(* CODESYS project refactoreddoworking.project
   CompiledLibraryCompatibilityVersion: LeadSysStudio V3.5 SP15 Patch 4
   Title: MC500_EtherCAT_axis_motion

Project tree, tasks and I/O mapping:
  Device : MC508, Leadshine Technology Co., Ltd., order no. 508101, version 3.5.15.40
      settings: RetainMode = 0; RetainStartAddr = 20480; RetainEndAddr = 524288; RetainSize = 524288
    application Application
      libraries: Standard, * (System); LS_ModbusMasterlib, 0.0.0.2 (Leadshine Technology Co.Ltd)
      task MainTask (cyclic, interval 4000 µs, priority 1) calls EtherCAT_Master_Leadshine_A.EtherCAT_Task, PLC_PRG
      global variables GVL_Shared
      program MainSeq [SFC]: A_Idle, A_HomeXY, A_GridCalc, A_GriddleDwell, A_MoveToPick, A_Grip, A_MoveToPlace, A_Release, A_NextOrDone, A_Park, A_Wait, A_Settle, A_Error, A_Hold, A_ZDownPick, A_ZUp, A_ZDownPlace, A_ZUpAfter, A_ZWait
      program PLC_PRG [CFC]
      program Inputs [LD]
      program Motion [CFC]
      function block GridCalc [ST]
    Resource Usage
    Network Configuration
      LocalBus Config
    Device Diagnose
    LocalBus_Master_Module : LocalBus Master, Leadshine Technology Co., Ltd., version 3.5.15.40
    High_Speed_IO_Module : High Speed IO, Leadshine Technology Co., Ltd., version 3.5.15.40
        unmapped channels: Genral_IO_IN, Genral_IO_Out
    SoftMotion General Axis Pool
    EtherCAT_Master_Leadshine_A : EtherCAT Master SoftMotion, 3S - Smart Software Solutions GmbH, version 3.5.15.30
        settings: NetworkName = 'ecat'; SelectNetworkByName = TRUE
      CS3E_D1008 : CS3E-D1008(COE), Leadshine Technology Co.,Ltd., order no. CS3E-D1008, version Revision=16#00000001
          settings: DC sync0 cycletime = 4000; DC sync1 cycletime = 4000; Number of SDO = 6; Homing method.Index = 16#6098; Homing method.Subindex = 16#00; Homing method.Value = 17; Homing method.Size = 8; Homing method.AbortIfError = FALSE; Homing method.JumpToLine = FALSE; Homing method.Line = 0; Homing method.CompleteAccess = FALSE; Homing velocity (fast).Index = 16#6099; Homing velocity (fast).Subindex = 16#01; Homing velocity (fast).Value = 2000; Homing velocity (fast).Size = 32; Homing velocity (fast).AbortIfError = FALSE; Homing velocity (fast).JumpToLine = FALSE; Homing velocity (fast).Line = 0; Homing velocity (fast).CompleteAccess = FALSE; Homing velocity (slow).Index = 16#6099; Homing velocity (slow).Subindex = 16#02; Homing velocity (slow).Value = 300; Homing velocity (slow).Size = 32; Homing velocity (slow).AbortIfError = FALSE; Homing velocity (slow).JumpToLine = FALSE; Homing velocity (slow).Line = 0; Homing velocity (slow).CompleteAccess = FALSE; Homing acceleration.Index = 16#609A; Homing acceleration.Subindex = 16#00; Homing acceleration.Value = 5000; Homing acceleration.Size = 32; Homing acceleration.AbortIfError = FALSE; Homing acceleration.JumpToLine = FALSE; Homing acceleration.Line = 0; Homing acceleration.CompleteAccess = FALSE; Homing offset.Index = 16#607C; Homing offset.Subindex = 16#00; Homing offset.Value = 0; Homing offset.Size = 32; Homing offset.AbortIfError = FALSE;
            Homing offset.JumpToLine = FALSE; Homing offset.Line = 0; Homing offset.CompleteAccess = FALSE
          input  yAxis_LastError : UINT  // Last Error Code
          unmapped channels: Control Word, Profile Target Position, Touch Probe Function, Status Word, Modes of Operation display, Position Actual Value, Touch Probe Status, Touch Probe 1 Positive Value, Digital Inputs
        yAxis : Axis, 3S - Smart Software Solutions GmbH, order no. 0, version 4.6.1.0
            settings: wDriveID = 0; dwRatioTechUnitsDenom = 20; eRampType = 3; Number of pulses for one revolution = 4000; The displacement for one revolution of the workbench = 100; Gear ratio molecule = 10; Gear ratio denominator = 10; Home velocity = 100; Home Creep speed = 15.000; Home acceleration = 250; Home position offset = 0; Home velocitySDO = 2000; Home Creep speedSDO = 300; Home position offsetSDO = 0; ScalingIncs = 4000; AdrOffset_8010 = 16; BitOffset_8010 = 0; BitLength_8010 = 16; Address_8010 = '%QW8'; Type_8010 = 'UINT'; AddressPointer_8010 = ADR(%QW8); AdrOffset_8020 = 20; BitOffset_8020 = 0; BitLength_8020 = 32; Address_8020 = '%QD5'; Type_8020 = 'DINT'; AddressPointer_8020 = ADR(%QD5); AdrOffset_8030 = 4294967295; BitOffset_8030 = 0; BitLength_8030 = 0; Address_8030 = ''; Type_8030 = ''; AddressPointer_8030 = 0; AdrOffset_8040 = 4294967295; BitOffset_8040 = 0; BitLength_8040 = 0; Address_8040 = ''; Type_8040 = ''; AddressPointer_8040 = 0; AdrOffset_8050 = 4294967295;
              BitOffset_8050 = 0; BitLength_8050 = 0; Address_8050 = ''; Type_8050 = ''; AddressPointer_8050 = 0; AdrOffset_8060 = 24; BitOffset_8060 = 0; BitLength_8060 = 16; Address_8060 = '%QW12'; Type_8060 = 'UINT'; AddressPointer_8060 = ADR(%QW12); AdrOffset_8070 = 4294967295; BitOffset_8070 = 0; BitLength_8070 = 0; Address_8070 = ''; Type_8070 = ''; AddressPointer_8070 = 0; AdrOffset_8080 = 4294967295; BitOffset_8080 = 0; BitLength_8080 = 0; Address_8080 = ''; Type_8080 = ''; AddressPointer_8080 = 0; AdrOffset_8090 = 4294967295; BitOffset_8090 = 0; BitLength_8090 = 0; Address_8090 = ''; Type_8090 = ''; AddressPointer_8090 = 0; AdrOffset_8510 = 30; BitOffset_8510 = 0; BitLength_8510 = 16; Address_8510 = '%IW15'; Type_8510 = 'UINT'; AddressPointer_8510 = ADR(%IW15); AdrOffset_8520 = 36; BitOffset_8520 = 0; BitLength_8520 = 32; Address_8520 = '%ID9'; Type_8520 = 'DINT';
              AddressPointer_8520 = ADR(%ID9); AdrOffset_8530 = 4294967295; BitOffset_8530 = 0; BitLength_8530 = 0; Address_8530 = ''; Type_8530 = ''; AddressPointer_8530 = 0; AdrOffset_8540 = 4294967295; BitOffset_8540 = 0; BitLength_8540 = 0; Address_8540 = ''; Type_8540 = ''; AddressPointer_8540 = 0; AdrOffset_8550 = 32; BitOffset_8550 = 0; BitLength_8550 = 8; Address_8550 = '%IB32'; Type_8550 = 'SINT'; AddressPointer_8550 = ADR(%IB32); AdrOffset_8560 = 48; BitOffset_8560 = 0; BitLength_8560 = 32; Address_8560 = '%ID12'; Type_8560 = 'UDINT'; AddressPointer_8560 = ADR(%ID12); AdrOffset_8570 = 40; BitOffset_8570 = 0; BitLength_8570 = 16; Address_8570 = '%IW20'; Type_8570 = 'UINT'; AddressPointer_8570 = ADR(%IW20); AdrOffset_8580 = 44; BitOffset_8580 = 0; BitLength_8580 = 32; Address_8580 = '%ID11'; Type_8580 = 'DINT'; AddressPointer_8580 = ADR(%ID11); AdrOffset_8590 = 4294967295; BitOffset_8590 = 0; BitLength_8590 = 0;
              Address_8590 = ''; Type_8590 = ''; AddressPointer_8590 = 0; AdrOffset_8600 = 4294967295; BitOffset_8600 = 0; BitLength_8600 = 0; Address_8600 = ''; Type_8600 = ''; AddressPointer_8600 = 0; AdrOffset_8600 = 4294967295; BitOffset_8600 = 0; BitLength_8600 = 0; Address_8610 = ''; Type_8610 = ''; AddressPointer_8610 = 0; AdrOffset_8620 = 4294967295; BitOffset_8620 = 0; BitLength_8620 = 0; Address_8620 = ''; Type_8620 = ''; AddressPointer_8620 = 0; Home accelerationSDO = 5000
      CS3E_D1008_1 : CS3E-D1008(COE), Leadshine Technology Co.,Ltd., order no. CS3E-D1008, version Revision=16#00000001
          settings: DC sync0 cycletime = 4000; DC sync1 cycletime = 4000; Number of SDO = 6; Homing method.Index = 16#6098; Homing method.Subindex = 16#00; Homing method.Value = 17; Homing method.Size = 8; Homing method.AbortIfError = FALSE; Homing method.JumpToLine = FALSE; Homing method.Line = 0; Homing method.CompleteAccess = False; Homing velocity (fast).Index = 16#6099; Homing velocity (fast).Subindex = 16#01; Homing velocity (fast).Value = 2000; Homing velocity (fast).Size = 32; Homing velocity (fast).AbortIfError = FALSE; Homing velocity (fast).JumpToLine = FALSE; Homing velocity (fast).Line = 0; Homing velocity (fast).CompleteAccess = False; Homing velocity (slow).Index = 16#6099; Homing velocity (slow).Subindex = 16#02; Homing velocity (slow).Value = 300; Homing velocity (slow).Size = 32; Homing velocity (slow).AbortIfError = FALSE; Homing velocity (slow).JumpToLine = FALSE; Homing velocity (slow).Line = 0; Homing velocity (slow).CompleteAccess = False; Homing acceleration.Index = 16#609A; Homing acceleration.Subindex = 16#00; Homing acceleration.Value = 5000; Homing acceleration.Size = 32; Homing acceleration.AbortIfError = FALSE; Homing acceleration.JumpToLine = FALSE; Homing acceleration.Line = 0; Homing acceleration.CompleteAccess = False; Homing offset.Index = 16#607C; Homing offset.Subindex = 16#00; Homing offset.Value = 0; Homing offset.Size = 32; Homing offset.AbortIfError = FALSE;
            Homing offset.JumpToLine = FALSE; Homing offset.Line = 0; Homing offset.CompleteAccess = False
          input  XAXIS_LastError : UINT  // Last Error Code
          unmapped channels: Control Word, Profile Target Position, Touch Probe Function, Status Word, Modes of Operation display, Position Actual Value, Touch Probe Status, Touch Probe 1 Positive Value, Digital Inputs
        XAXIS : Axis, 3S - Smart Software Solutions GmbH, order no. 0, version 4.6.1.0
            settings: dwRatioTechUnitsDenom = 20; Commisioning.smci.Distance = 110; Commisioning.smci.Velocity = 100; Gear ratio molecule = 500; Gear ratio denominator = 500; Home velocity = 100; Home Creep speed = 15; Home acceleration = 250; Home position offset = 0; Home velocitySDO = 2000; Home Creep speedSDO = 300; Home position offsetSDO = 0; ScalingIncs = 4000; InvertDirection = False; AdrOffset_8010 = 4; BitOffset_8010 = 0; BitLength_8010 = 16; Address_8010 = '%QW2'; Type_8010 = 'UINT'; AddressPointer_8010 = ADR(%QW2); AdrOffset_8020 = 8; BitOffset_8020 = 0; BitLength_8020 = 32; Address_8020 = '%QD2'; Type_8020 = 'DINT'; AddressPointer_8020 = ADR(%QD2); AdrOffset_8030 = 4294967295; BitOffset_8030 = 0; BitLength_8030 = 0; Address_8030 = ''; Type_8030 = ''; AddressPointer_8030 = 0; AdrOffset_8040 = 4294967295; BitOffset_8040 = 0; BitLength_8040 = 0; Address_8040 = ''; Type_8040 = ''; AddressPointer_8040 = 0; AdrOffset_8050 = 4294967295; BitOffset_8050 = 0;
              BitLength_8050 = 0; Address_8050 = ''; Type_8050 = ''; AddressPointer_8050 = 0; AdrOffset_8060 = 12; BitOffset_8060 = 0; BitLength_8060 = 16; Address_8060 = '%QW6'; Type_8060 = 'UINT'; AddressPointer_8060 = ADR(%QW6); AdrOffset_8070 = 4294967295; BitOffset_8070 = 0; BitLength_8070 = 0; Address_8070 = ''; Type_8070 = ''; AddressPointer_8070 = 0; AdrOffset_8080 = 4294967295; BitOffset_8080 = 0; BitLength_8080 = 0; Address_8080 = ''; Type_8080 = ''; AddressPointer_8080 = 0; AdrOffset_8090 = 4294967295; BitOffset_8090 = 0; BitLength_8090 = 0; Address_8090 = ''; Type_8090 = ''; AddressPointer_8090 = 0; AdrOffset_8510 = 6; BitOffset_8510 = 0; BitLength_8510 = 16; Address_8510 = '%IW3'; Type_8510 = 'UINT'; AddressPointer_8510 = ADR(%IW3); AdrOffset_8520 = 12; BitOffset_8520 = 0; BitLength_8520 = 32; Address_8520 = '%ID3'; Type_8520 = 'DINT'; AddressPointer_8520 = ADR(%ID3);
              AdrOffset_8530 = 4294967295; BitOffset_8530 = 0; BitLength_8530 = 0; Address_8530 = ''; Type_8530 = ''; AddressPointer_8530 = 0; AdrOffset_8540 = 4294967295; BitOffset_8540 = 0; BitLength_8540 = 0; Address_8540 = ''; Type_8540 = ''; AddressPointer_8540 = 0; AdrOffset_8550 = 8; BitOffset_8550 = 0; BitLength_8550 = 8; Address_8550 = '%IB8'; Type_8550 = 'SINT'; AddressPointer_8550 = ADR(%IB8); AdrOffset_8560 = 24; BitOffset_8560 = 0; BitLength_8560 = 32; Address_8560 = '%ID6'; Type_8560 = 'UDINT'; AddressPointer_8560 = ADR(%ID6); AdrOffset_8570 = 16; BitOffset_8570 = 0; BitLength_8570 = 16; Address_8570 = '%IW8'; Type_8570 = 'UINT'; AddressPointer_8570 = ADR(%IW8); AdrOffset_8580 = 20; BitOffset_8580 = 0; BitLength_8580 = 32; Address_8580 = '%ID5'; Type_8580 = 'DINT'; AddressPointer_8580 = ADR(%ID5); AdrOffset_8590 = 4294967295; BitOffset_8590 = 0; BitLength_8590 = 0; Address_8590 = '';
              Type_8590 = ''; AddressPointer_8590 = 0; AdrOffset_8600 = 4294967295; BitOffset_8600 = 0; BitLength_8600 = 0; Address_8600 = ''; Type_8600 = ''; AddressPointer_8600 = 0; AdrOffset_8600 = 4294967295; BitOffset_8600 = 0; BitLength_8600 = 0; Address_8610 = ''; Type_8610 = ''; AddressPointer_8610 = 0; AdrOffset_8620 = 4294967295; BitOffset_8620 = 0; BitLength_8620 = 0; Address_8620 = ''; Type_8620 = ''; AddressPointer_8620 = 0; Home accelerationSDO = 5000
    ModbusTCP_Slave_Device : Modbus TCP Slave, Leadshine Technology Co., Ltd., version 00.00.00.10
*)

// Device/Application/GVL_Shared
// =====================================================================
// GVL  "GVL_Shared"  — globals shared across the LD / CFC / SFC / ST POUs
// (Splitting one POU into four means the formerly-local VARs become globals
//  grouped by owner. Comment // [owner->reader] shows the data direction.)
// =====================================================================
VAR_GLOBAL
    // ---- AXIS REFERENCES (declared in your hardware config) ----
    // XAXIS, yAxis : AXIS_REF;   // already exist in the project

    // ============ COMMAND FLAGS : LD (Inputs) -> SFC ============
    pending_start   : BOOL := FALSE;
    
    pending_resume  : BOOL := FALSE;
   
    hmi_start       : BOOL := FALSE;   // HMI write
   
    sw_a            : BOOL := FALSE;    // HMI/soft button A
    sw_b            : BOOL := FALSE;    // HMI/soft button B

    // ============ MOTION REQUESTS : SFC -> CFC (Motion) =========
    gMoveExec    : BOOL := FALSE;          // drive LS_MoveXY.Exec
    gHomeExec    : BOOL := FALSE;          // drive MC_Home_1/2.Execute
    gStopExec    : BOOL := FALSE;          // drive MC_Stop_1/2.Execute
    TargetXY     : ARRAY[0..1] OF LREAL := [0.0, 0.0];
    drive_enable : BOOL := TRUE;           // MC_Power_*.Enable (set by Inputs/Pause)

    // ============ MOTION STATUS : CFC (Motion) -> SFC ===========
    gPowerOK   : BOOL := FALSE;            // MC_Power_1.Status AND MC_Power_2.Status
    gMoveDone  : BOOL := FALSE;            // LS_MoveXY.Done
    gMoveErr   : BOOL := FALSE;            // LS_MoveXY.Error 
    gMoveBusy  : BOOL := FALSE;            // LS_MoveXY.Busy
    gHomeDone  : BOOL := FALSE;            // MC_Home_1.Done AND MC_Home_2.Done
    gStopDone  : BOOL := FALSE;            // MC_Stop_1.Done AND MC_Stop_2.Done

    // ============ END EFFECTOR + STOP TUNING ====================
    end_effector AT %QX1.4 : BOOL := FALSE;   // LD coil
    QUICK_STOP_DECEL : LREAL := 3000.0;

    // ============ Z AXIS — MODBUS I/O (CS2RS-D1008) =============


    // ============ TRAY / GRID CONFIG (read by GridCalc) ========
    PICK_BASE_X    : LREAL := 145.0;
    PICK_BASE_Y    : LREAL := 45.0;
    PICK_SPACING_X : LREAL := 80.0;
    PICK_SPACING_Y : LREAL := 80.0;
    PLACE_BASE_X   : LREAL := 740.0;
    PLACE_BASE_Y   : LREAL := 116.0;
    PLACE_OFFSET_X : ARRAY[0..5] OF LREAL := [0.0, 70.0, -70.0, 70.0, -70.0, 0.0];
    PLACE_OFFSET_Y : ARRAY[0..5] OF LREAL := [0.0, 66.0, 66.0, 143.0, 143.0, 210.0];
    TRAY_COLS           : INT := 6;
    TRAY_ROWS           : INT := 4;
    TOTAL_PATTIES       : INT := 24;
    PATTIES_PER_GRIDDLE : INT := 6;
    GRIDDLE_COUNT       : INT := 4;

    // ============ GRID RESULTS (GridCalc -> SFC) ===============
    patty_index   : INT := 0;
    current_col   : INT := 0;
    current_row   : INT := 0;
    griddle_index : INT := 0;
    slot_index    : INT := 0;
    pick_x  : LREAL := 0.0;   pick_y  : LREAL := 0.0;
    place_x : LREAL := 0.0;   place_y : LREAL := 0.0;

    // ============ MODE / BOOKKEEPING ===========================
    TEST_LOOP_MODE : BOOL := TRUE;
    cycle_count    : UDINT := 0;
    cycle_complete : BOOL := FALSE;
    cycle_active   : BOOL := FALSE;
    paused         : BOOL := FALSE;
   
    
    

    // ============ TIMING CONSTANTS =============================

   
    XY_HOME_WAIT   : INT := 7500;
    xy_home_timer  : INT := 0;
	
	stop_request  : BOOL := FALSE;   // CYCLE-stop request (operator Stop button)
	holding       : BOOL := FALSE;   // TRUE while parked & held
	pending_reset : BOOL := FALSE;
	hmi_stop      : BOOL := FALSE;
	hmi_reset     : BOOL := FALSE;
	
	
	Z_DO_Down    AT %QX1.5 : BOOL := FALSE;   // pulse -> down path
	Z_InPos      AT %IX1.0 : BOOL;            // SO1 INP = positioning complete
	z_saw_moving : BOOL := FALSE;
	Z_Alarm AT %IX1.1 : BOOL;   // SO3 ALM (check polarity)
	z_wait_count   : INT  := 0;
    Z_MOVE_TIMEOUT : INT  := 2500;
	
	state : INT := 0;
	Z_Disable AT %QX1.3 : BOOL := FALSE;   // TRUE = disable Z drive; FALSE (default) = enabled
	Z_Trig AT %QX1.6 : BOOL := FALSE; 
	xy_moving : BOOL := FALSE;
	np_done : BOOL := FALSE;
END_VAR

// Device/Application/PLC_PRG
PROGRAM PLC_PRG
VAR
   
END_VAR

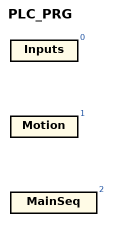
Inputs();
Motion();
MainSeq();

END_PROGRAM

// Device/Application/Inputs
PROGRAM Inputs
VAR
	btn_a AT %IX0.0 : BOOL;
    btn_b AT %IX0.1 : BOOL;
    rt_a : R_TRIG;
    rt_b : R_TRIG;
    edgeA : BOOL;                  
	edgeB : BOOL;
	btn_reset AT %IX0.2 : BOOL;   // physical Reset (wire later)
	rt_reset  : R_TRIG;
	edgeReset : BOOL;
END_VAR

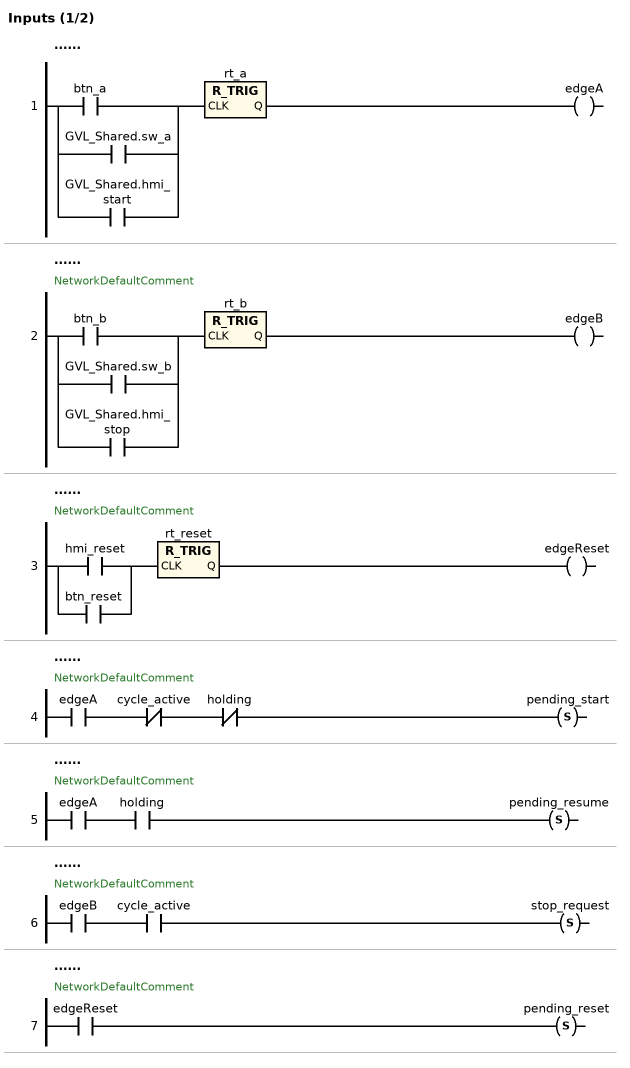
// NETWORK 1: ......
rt_a(CLK := btn_a OR GVL_Shared.sw_a OR GVL_Shared.hmi_start); // R_TRIG
edgeA := rt_a.Q;

// NETWORK 2: ......
// NetworkDefaultComment
rt_b(CLK := btn_b OR GVL_Shared.sw_b OR GVL_Shared.hmi_stop); // R_TRIG
edgeB := rt_b.Q;

// NETWORK 3: ......
// NetworkDefaultComment
rt_reset(CLK := hmi_reset OR btn_reset); // R_TRIG
edgeReset := rt_reset.Q;

// NETWORK 4: ......
// NetworkDefaultComment
pending_start S= edgeA AND NOT cycle_active AND NOT holding;

// NETWORK 5: ......
// NetworkDefaultComment
pending_resume S= edgeA AND holding;

// NETWORK 6: ......
// NetworkDefaultComment
stop_request S= edgeB AND cycle_active;

// NETWORK 7: ......
// NetworkDefaultComment
pending_reset S= edgeReset;

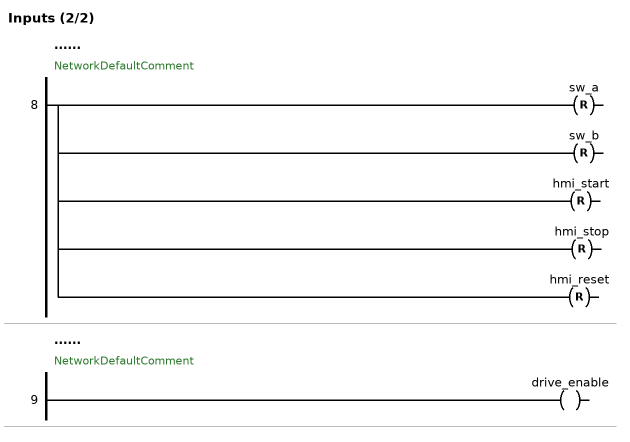
// NETWORK 8: ......
// NetworkDefaultComment
sw_a R= TRUE;
sw_b R= TRUE;
hmi_start R= TRUE;
hmi_stop R= TRUE;
hmi_reset R= TRUE;

// NETWORK 9: ......
// NetworkDefaultComment
drive_enable := TRUE;

END_PROGRAM

// Device/Application/Motion
PROGRAM Motion
VAR
	MC_Power_1: MC_Power;
	MC_Power_2: MC_Power;
	MC_Home_1: MC_Home;
	MC_Home_2: MC_Home;
	MC_Stop_1: MC_Stop;
	MC_Stop_2: MC_Stop;
	MC_Reset_1: MC_Reset;
	LS_MOVEXY: LS_2AxisLine;
	MC_Reset_2: MC_Reset;
END_VAR

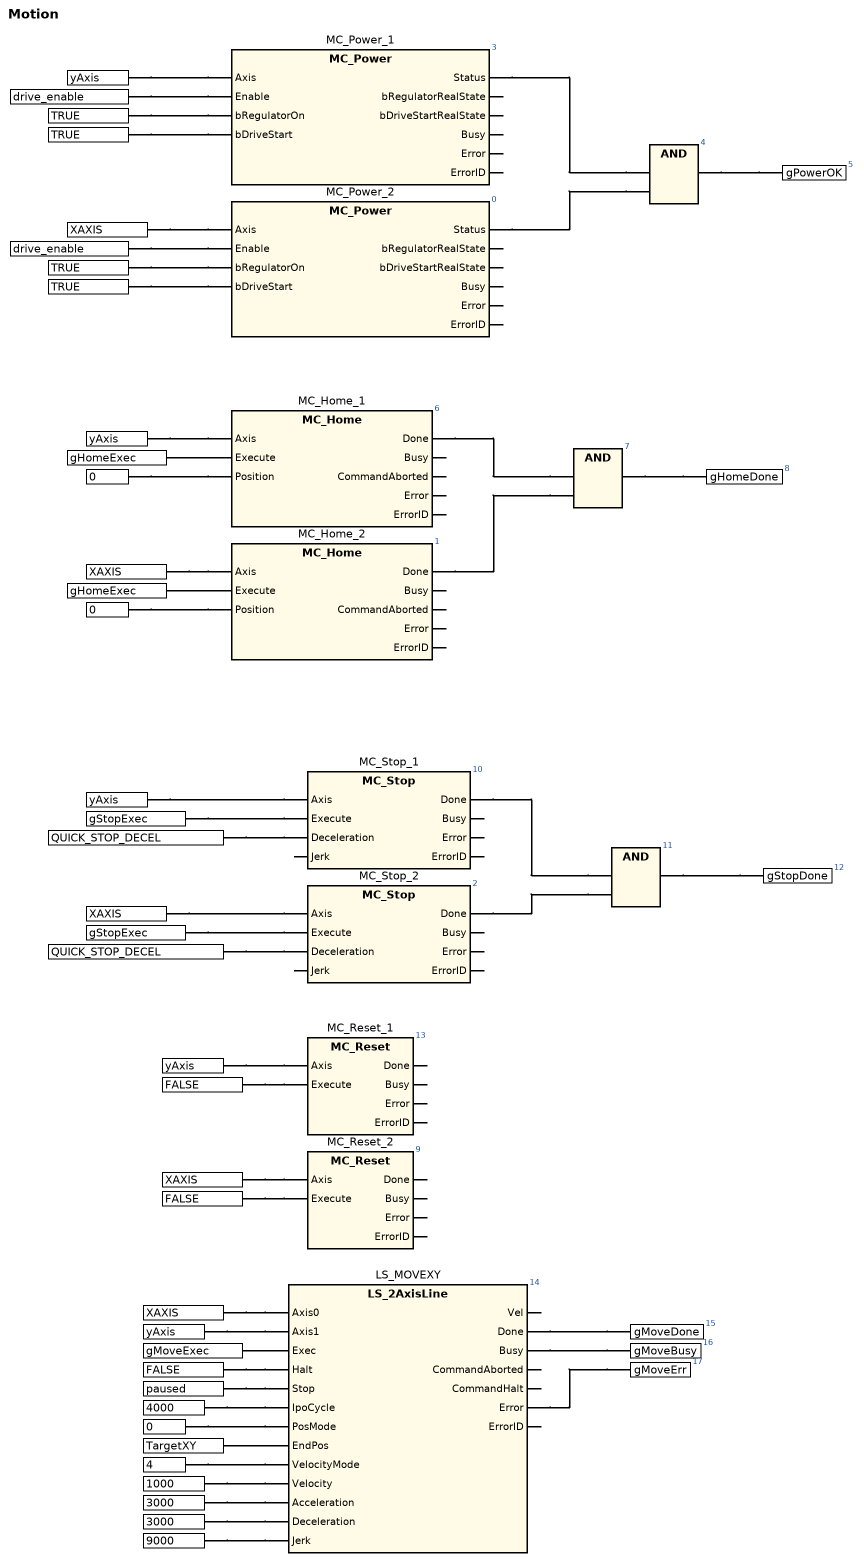
MC_Power_2(Axis := XAXIS, Enable := drive_enable, bRegulatorOn := TRUE, bDriveStart := TRUE); // MC_Power
MC_Home_2(Axis := XAXIS, Execute := gHomeExec, Position := 0); // MC_Home
MC_Stop_2(Axis := XAXIS, Execute := gStopExec, Deceleration := QUICK_STOP_DECEL); // MC_Stop
MC_Power_1(Axis := yAxis, Enable := drive_enable, bRegulatorOn := TRUE, bDriveStart := TRUE); // MC_Power
gPowerOK := MC_Power_1.Status AND MC_Power_2.Status;
MC_Home_1(Axis := yAxis, Execute := gHomeExec, Position := 0); // MC_Home
gHomeDone := MC_Home_1.Done AND MC_Home_2.Done;
MC_Reset_2(Axis := XAXIS, Execute := FALSE); // MC_Reset
MC_Stop_1(Axis := yAxis, Execute := gStopExec, Deceleration := QUICK_STOP_DECEL); // MC_Stop
gStopDone := MC_Stop_1.Done AND MC_Stop_2.Done;
MC_Reset_1(Axis := yAxis, Execute := FALSE); // MC_Reset
LS_MOVEXY(
    Axis0 := XAXIS,
    Axis1 := yAxis,
    Exec := gMoveExec,
    Halt := FALSE,
    Stop := paused,
    IpoCycle := 4000,
    PosMode := 0,
    EndPos := TargetXY,
    VelocityMode := 4,
    Velocity := 1000,
    Acceleration := 3000,
    Deceleration := 3000,
    Jerk := 9000); // LS_2AxisLine
gMoveDone := LS_MOVEXY.Done;
gMoveBusy := LS_MOVEXY.Busy;
gMoveErr := LS_MOVEXY.Error;

END_PROGRAM

// Device/Application/MainSeq
PROGRAM MainSeq
VAR
    // function-block instances this POU owns
    fbGrid  : GridCalc;        // grid math, called in A_GridCalc

    // step timers (local to MainSeq)
    griddle_dwell : TON;       // A_Error, A_GriddleDwell, A_Idle
    grip_timer    : TON;       // A_Grip, A_Release
    loop_dwell    : TON;       // A_Wait
   

    // time constants
    GRIP_TIME       : TIME := T#500MS;
    RELEASE_TIME    : TIME := T#500MS;
    GRIDDLE_DWELL_T : TIME := T#5S;
    LOOP_DWELL_T    : TIME := T#3S;
    
END_VAR

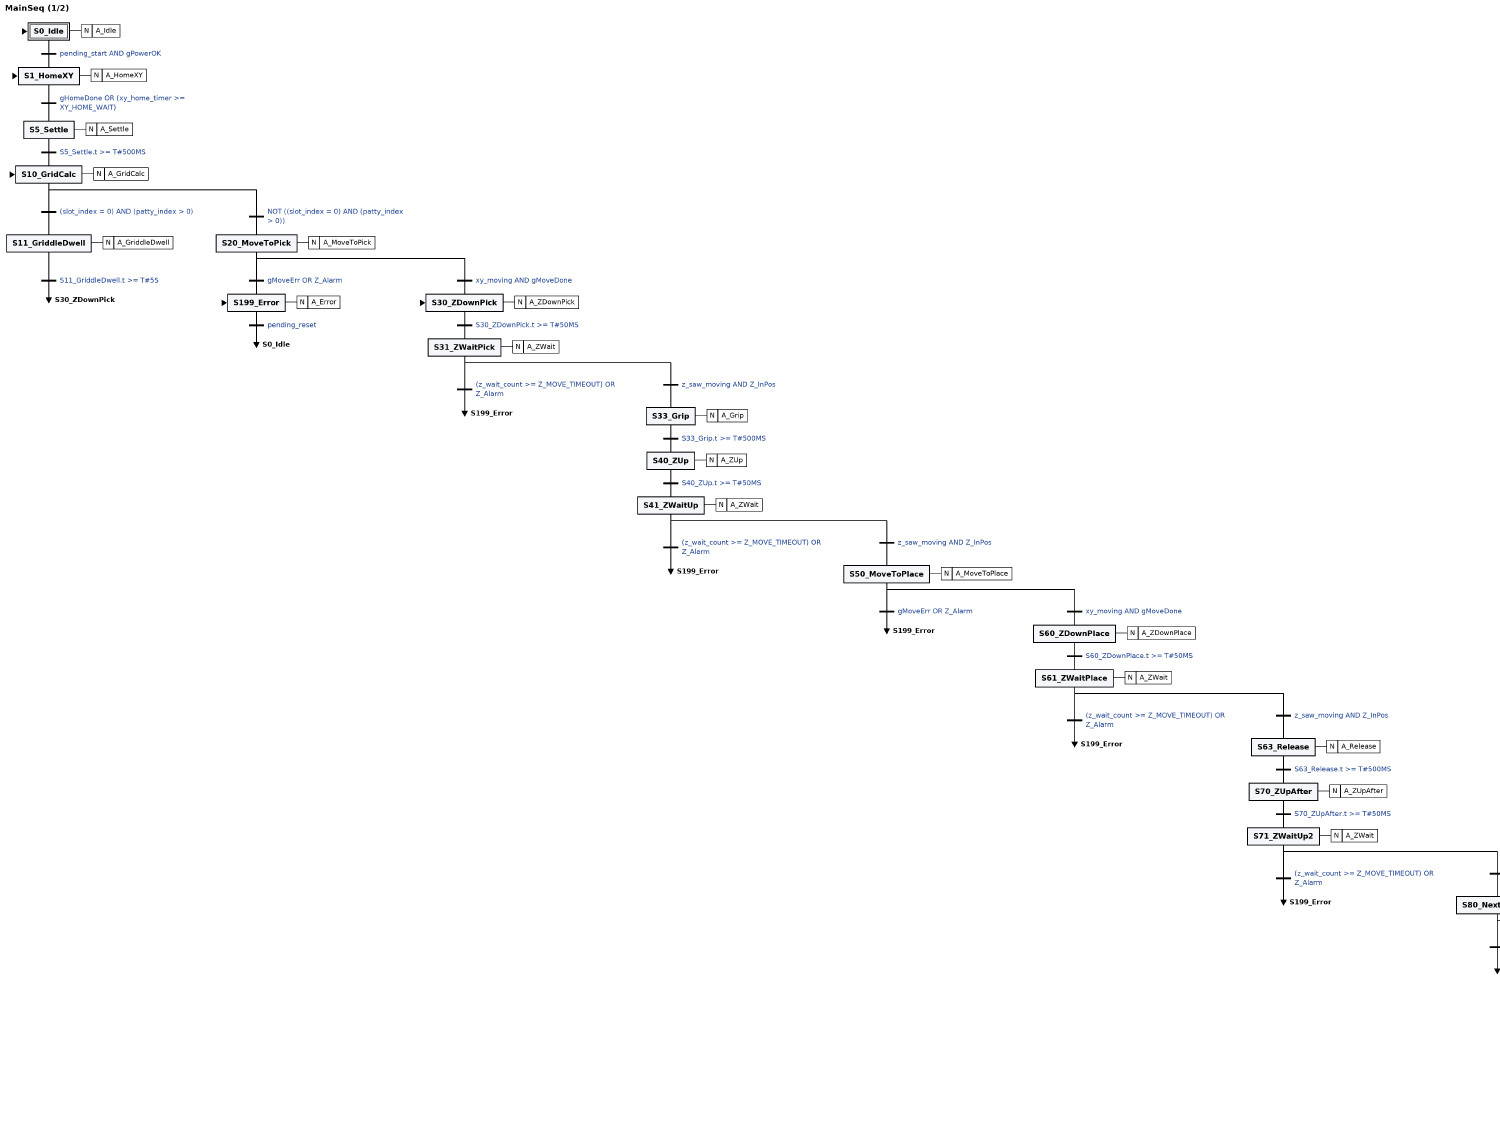
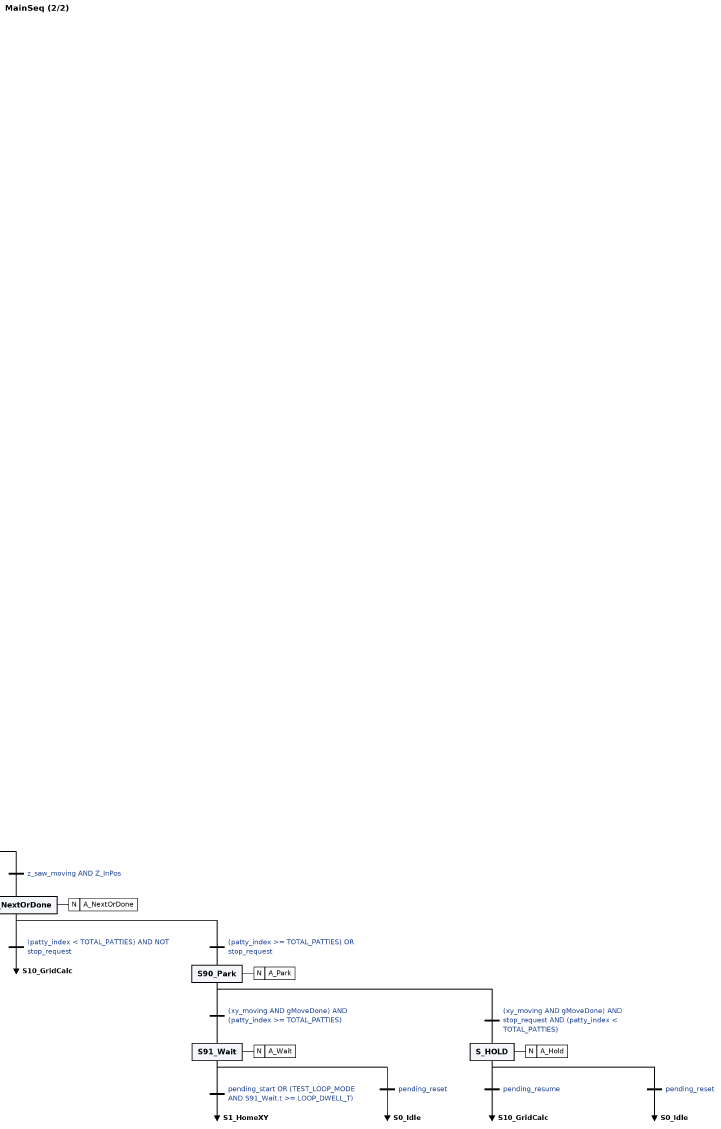
INITIAL_STEP S0_Idle:
    A_Idle(N);
END_STEP
TRANSITION FROM S0_Idle TO S1_HomeXY
    := pending_start AND gPowerOK;
END_TRANSITION
STEP S1_HomeXY:
    A_HomeXY(N);
END_STEP
TRANSITION FROM S1_HomeXY TO S5_Settle
    := gHomeDone OR (xy_home_timer >= XY_HOME_WAIT);
END_TRANSITION
STEP S5_Settle:
    A_Settle(N);
END_STEP
TRANSITION FROM S5_Settle TO S10_GridCalc
    := S5_Settle.t >= T#500MS;
END_TRANSITION
STEP S10_GridCalc:
    A_GridCalc(N);
END_STEP
TRANSITION FROM S10_GridCalc TO S11_GriddleDwell
    := (slot_index = 0) AND (patty_index > 0);
END_TRANSITION
STEP S11_GriddleDwell:
    A_GriddleDwell(N);
END_STEP
TRANSITION FROM S11_GriddleDwell TO S30_ZDownPick
    := S11_GriddleDwell.t >= T#5S;
END_TRANSITION
TRANSITION FROM S10_GridCalc TO S20_MoveToPick
    := NOT ((slot_index = 0) AND (patty_index > 0));
END_TRANSITION
STEP S20_MoveToPick:
    A_MoveToPick(N);
END_STEP
TRANSITION FROM S20_MoveToPick TO S199_Error
    := gMoveErr OR Z_Alarm;
END_TRANSITION
STEP S199_Error:
    A_Error(N);
END_STEP
TRANSITION FROM S199_Error TO S0_Idle
    := pending_reset;
END_TRANSITION
TRANSITION FROM S20_MoveToPick TO S30_ZDownPick
    := xy_moving AND gMoveDone;
END_TRANSITION
STEP S30_ZDownPick:
    A_ZDownPick(N);
END_STEP
TRANSITION FROM S30_ZDownPick TO S31_ZWaitPick
    := S30_ZDownPick.t >= T#50MS;
END_TRANSITION
STEP S31_ZWaitPick:
    A_ZWait(N);
END_STEP
TRANSITION FROM S31_ZWaitPick TO S199_Error
    := (z_wait_count >= Z_MOVE_TIMEOUT) OR Z_Alarm;
END_TRANSITION
TRANSITION FROM S31_ZWaitPick TO S33_Grip
    := z_saw_moving AND Z_InPos;
END_TRANSITION
STEP S33_Grip:
    A_Grip(N);
END_STEP
TRANSITION FROM S33_Grip TO S40_ZUp
    := S33_Grip.t >= T#500MS;
END_TRANSITION
STEP S40_ZUp:
    A_ZUp(N);
END_STEP
TRANSITION FROM S40_ZUp TO S41_ZWaitUp
    := S40_ZUp.t >= T#50MS;
END_TRANSITION
STEP S41_ZWaitUp:
    A_ZWait(N);
END_STEP
TRANSITION FROM S41_ZWaitUp TO S199_Error
    := (z_wait_count >= Z_MOVE_TIMEOUT) OR Z_Alarm;
END_TRANSITION
TRANSITION FROM S41_ZWaitUp TO S50_MoveToPlace
    := z_saw_moving AND Z_InPos;
END_TRANSITION
STEP S50_MoveToPlace:
    A_MoveToPlace(N);
END_STEP
TRANSITION FROM S50_MoveToPlace TO S199_Error
    := gMoveErr OR Z_Alarm;
END_TRANSITION
TRANSITION FROM S50_MoveToPlace TO S60_ZDownPlace
    := xy_moving AND gMoveDone;
END_TRANSITION
STEP S60_ZDownPlace:
    A_ZDownPlace(N);
END_STEP
TRANSITION FROM S60_ZDownPlace TO S61_ZWaitPlace
    := S60_ZDownPlace.t >= T#50MS;
END_TRANSITION
STEP S61_ZWaitPlace:
    A_ZWait(N);
END_STEP
TRANSITION FROM S61_ZWaitPlace TO S199_Error
    := (z_wait_count >= Z_MOVE_TIMEOUT) OR Z_Alarm;
END_TRANSITION
TRANSITION FROM S61_ZWaitPlace TO S63_Release
    := z_saw_moving AND Z_InPos;
END_TRANSITION
STEP S63_Release:
    A_Release(N);
END_STEP
TRANSITION FROM S63_Release TO S70_ZUpAfter
    := S63_Release.t >= T#500MS;
END_TRANSITION
STEP S70_ZUpAfter:
    A_ZUpAfter(N);
END_STEP
TRANSITION FROM S70_ZUpAfter TO S71_ZWaitUp2
    := S70_ZUpAfter.t >= T#50MS;
END_TRANSITION
STEP S71_ZWaitUp2:
    A_ZWait(N);
END_STEP
TRANSITION FROM S71_ZWaitUp2 TO S199_Error
    := (z_wait_count >= Z_MOVE_TIMEOUT) OR Z_Alarm;
END_TRANSITION
TRANSITION FROM S71_ZWaitUp2 TO S80_NextOrDone
    := z_saw_moving AND Z_InPos;
END_TRANSITION
STEP S80_NextOrDone:
    A_NextOrDone(N);
END_STEP
TRANSITION FROM S80_NextOrDone TO S10_GridCalc
    := (patty_index < TOTAL_PATTIES) AND NOT stop_request;
END_TRANSITION
TRANSITION FROM S80_NextOrDone TO S90_Park
    := (patty_index >= TOTAL_PATTIES) OR stop_request;
END_TRANSITION
STEP S90_Park:
    A_Park(N);
END_STEP
TRANSITION FROM S90_Park TO S91_Wait
    := (xy_moving AND gMoveDone) AND (patty_index >= TOTAL_PATTIES);
END_TRANSITION
TRANSITION FROM S90_Park TO S_HOLD
    := (xy_moving AND gMoveDone) AND stop_request AND (patty_index < TOTAL_PATTIES);
END_TRANSITION
STEP S_HOLD:
    A_Hold(N);
END_STEP
TRANSITION FROM S_HOLD TO S10_GridCalc
    := pending_resume;
END_TRANSITION
TRANSITION FROM S_HOLD TO S0_Idle
    := pending_reset;
END_TRANSITION
STEP S91_Wait:
    A_Wait(N);
END_STEP
TRANSITION FROM S91_Wait TO S1_HomeXY
    := pending_start OR (TEST_LOOP_MODE AND S91_Wait.t >= LOOP_DWELL_T);
END_TRANSITION
TRANSITION FROM S91_Wait TO S0_Idle
    := pending_reset;
END_TRANSITION

ACTION A_Idle:
state := 0;
cycle_complete := FALSE;  cycle_active := FALSE;  paused := FALSE;
end_effector := FALSE;
z_wait_count := 0;        xy_home_timer := 0;
griddle_index := 0;       slot_index := 0;
griddle_dwell(IN := FALSE);
gMoveExec := FALSE;  gHomeExec := FALSE;  gStopExec := FALSE;
xy_moving := FALSE;  np_done := FALSE;          // <-- add np_done here
Z_DO_Down := FALSE;  Z_Trig := FALSE;
stop_request := FALSE;  holding := FALSE;  pending_reset := FALSE;
END_ACTION

ACTION A_HomeXY:
state := 1;
IF NOT cycle_active THEN
    pending_start := FALSE;        // ← drop the pending_restart line
    patty_index := 0;
	np_done := FALSE;  
  	cycle_active := TRUE;
END_IF
gHomeExec := TRUE;
xy_home_timer := xy_home_timer + 1;
IF gHomeDone OR (xy_home_timer >= XY_HOME_WAIT) THEN
    gHomeExec := FALSE;  xy_home_timer := 0;  z_wait_count := 0;
END_IF
END_ACTION

ACTION A_GridCalc:
state := 10;
IF holding THEN
    holding := FALSE;
    stop_request := FALSE;
    pending_resume := FALSE;
    cycle_active := TRUE;
END_IF
fbGrid(idx := patty_index);
END_ACTION

ACTION A_GriddleDwell:
state := 11;
griddle_dwell(IN := TRUE, PT := GRIDDLE_DWELL_T);
TargetXY[0] := pick_x;  TargetXY[1] := pick_y;     // travel to pick during rotation
gMoveExec := TRUE;
IF gMoveBusy OR NOT gMoveDone THEN xy_moving := TRUE; END_IF
IF griddle_dwell.Q THEN griddle_dwell(IN := FALSE); END_IF
END_ACTION

ACTION A_MoveToPick:
state := 20;
TargetXY[0] := pick_x;  TargetXY[1] := pick_y;
gMoveExec := TRUE;
IF gMoveBusy OR NOT gMoveDone THEN xy_moving := TRUE; END_IF
END_ACTION

ACTION A_Grip:
state := 33;
end_effector := TRUE;
END_ACTION

ACTION A_MoveToPlace:
state := 50;
TargetXY[0] := place_x;  TargetXY[1] := place_y;
gMoveExec := TRUE;
IF gMoveBusy OR NOT gMoveDone THEN xy_moving := TRUE; END_IF
END_ACTION

ACTION A_Release:
state := 63;
end_effector := FALSE;
END_ACTION

ACTION A_NextOrDone:
state := 80;
IF NOT np_done THEN
    patty_index := patty_index + 1;
    np_done := TRUE;
END_IF
END_ACTION

ACTION A_Park:
state := 90;
TargetXY[0] := 50.0;  TargetXY[1] := 50.0;
gMoveExec := TRUE;
IF gMoveBusy OR NOT gMoveDone THEN xy_moving := TRUE; END_IF
IF (xy_moving AND gMoveDone) OR gMoveErr THEN
    cycle_active := FALSE;
    IF patty_index >= TOTAL_PATTIES THEN
        cycle_complete := TRUE;
        cycle_count := cycle_count + 1;
    END_IF
END_IF
END_ACTION

ACTION A_Wait:
state := 91;
gMoveExec := FALSE;  xy_moving := FALSE;      // release the park move
np_done := FALSE;                             // arm patty counter for next run
END_ACTION

ACTION A_Settle:
state := 5;
  gHomeExec := FALSE;
  gMoveExec := FALSE;
END_ACTION

ACTION A_Error:
state := 199;
gMoveExec := FALSE;
gHomeExec := FALSE;
gStopExec := FALSE;
end_effector := FALSE;
griddle_dwell(IN := FALSE);
 Z_DO_Down := FALSE;
END_ACTION

ACTION A_Hold:
state := 95;
holding := TRUE;
cycle_active := FALSE;
gMoveExec := FALSE;  xy_moving := FALSE;
END_ACTION

ACTION A_ZDownPick:
state := 30;
gMoveExec := FALSE;  xy_moving := FALSE;     // release the pick move
Z_DO_Down := TRUE;   Z_Trig := FALSE;        // select down path, CTRG low
z_saw_moving := FALSE;  z_wait_count := 0;
END_ACTION

ACTION A_ZUp:
state:=40; Z_DO_Down := FALSE; Z_Trig := FALSE; z_saw_moving:=FALSE; z_wait_count:=0;
END_ACTION

ACTION A_ZDownPlace:
state := 60;
gMoveExec := FALSE;  xy_moving := FALSE;     // release the place move
Z_DO_Down := TRUE;   Z_Trig := FALSE;
z_saw_moving := FALSE;  z_wait_count := 0;
END_ACTION

ACTION A_ZUpAfter:
state := 70;
gMoveExec := FALSE;  xy_moving := FALSE;     // (if you added these — keep)
Z_DO_Down := FALSE;  Z_Trig := FALSE;
z_saw_moving := FALSE;  z_wait_count := 0;
np_done := FALSE;                            // arm the one-shot for S80
END_ACTION

ACTION A_ZWait:
Z_Trig := TRUE;                 // rising edge (address was set last step) -> executes selected path
z_wait_count := z_wait_count + 1;
IF NOT Z_InPos THEN
    z_saw_moving := TRUE;
END_IF
END_ACTION

END_PROGRAM

// Device/Application/GridCalc
// ---- DECLARATION pane ----
FUNCTION_BLOCK GridCalc
VAR_INPUT
    idx : INT;            // = patty_index
END_VAR
// (all the PICK_*/PLACE_*/result vars live in GVL_Shared)


current_row := idx / TRAY_COLS;
current_col := idx MOD TRAY_COLS;
pick_x := PICK_BASE_X + INT_TO_LREAL(current_col) * PICK_SPACING_X;
pick_y := PICK_BASE_Y + INT_TO_LREAL(current_row) * PICK_SPACING_Y;
 
griddle_index := idx / PATTIES_PER_GRIDDLE;
slot_index    := idx MOD PATTIES_PER_GRIDDLE;
place_x := PLACE_BASE_X + PLACE_OFFSET_X[slot_index];
place_y := PLACE_BASE_Y + PLACE_OFFSET_Y[slot_index];

END_FUNCTION_BLOCK
